{attribute 'qualified_only'}
{attribute 'strict'}
{attribute 'to_string'}
TYPE E_TransferState :
(
	Idle,
    Prepared,
    Requested,
    Accepted,
    WaitingContext,
    Ready,
    Transferring,
    LocalComplete,
    CommitPending,
    Committed,
    Aborting,
    Aborted,
    Error,
    RecoveryRequired
);
END_TYPE

(* stored: Version 1.1.0.1, ProductVersion 3.1.4026.18
   DUT E_TransferState: Id {87f5958e-bbdf-49d6-80cd-96b650d42eab} *)
